# EPICS IOC start-up script: examples/test/PSI/ep2624.iocsh
#- mXsXXX naming
require ecmccfg v7_RC1, "NAMING=mXsXXX"

#- add slaves
${SCRIPTEXEC} ${ecmccfg_DIR}addSlave.cmd, "HW_DESC=EP2624, SLAVE_ID=5"
